TYPE ST_PNOZEtherCATOut :
STRUCT
    stFeedback          : ST_SafetyFeedback;
    aSafetyFunctionOUT  : ARRAY[1..GVL_SafetyIO.UPPER_BOUND_SF] OF ST_SafetyFunctionOUT;
    aSubSystemOut       : ARRAY[1..GVL_SafetyIO.UPPER_BOUND_SS] OF ST_SubSystemOut;
    stSequenceOut       : ST_SequenceOut;
END_STRUCT
END_TYPE

(* stored: Version 1.1.0.1
   DUT ST_PNOZEtherCATOut: Id {2f65ec2d-5561-0256-2e54-58b3e165bd48} *)
